{attribute 'qualified_only'}
{attribute 'strict'}
TYPE EFeedbackMsgAttenuationELL18 :
(
	StateMsg := 1,
	PositionMsg := 10,
    IdMsg,
    CustomMsg
);
END_TYPE

(* stored: Version 1.1.0.1, ProductVersion 3.1.4024.10
   DUT EFeedbackMsgAttenuationELL18: Id {b98bd175-fb6a-46be-9412-7078cd2b2cd9} *)
